PROGRAM PRG_OPT_XPM
VAR
	bInit: BOOL :=TRUE;
	
	fb2AxesXPM: FB_2AxesTrans;
	bExecuteMotionXPM: BOOL :=TRUE;
	bMoveOkXPM: BOOL :=TRUE;
END_VAR

VAR CONSTANT
	rDistance	:REAL	:=	0.4;
END_VAR



IF bINIT THEN
	
	GVL_Main.M12.nBrakeMode := ENUM_StageBrakeMode.NO_BRAKE;
	GVL_Main.M12.bHardwareEnable := TRUE;
	GVL_Main.M12.bPowerSelf := TRUE;
	GVL_Main.M13.nBrakeMode := ENUM_StageBrakeMode.NO_BRAKE;
	GVL_Main.M13.bHardwareEnable := TRUE;
	GVL_Main.M13.bPowerSelf := TRUE;
	
		//
	GVL_Main.M12.nEnableMode := ENUM_StageEnableMode.DURING_MOTION ;
	GVL_Main.M13.nEnableMode := ENUM_StageEnableMode.DURING_MOTION ;

	bINIT := FALSE;
END_IF;

fb2AxesXPM(	i_DevName		:=	'OPT_XPM',
			stFirstAxis		:=	GVL_Main.M12,
			stSecondAxis	:=	GVL_Main.M13,
			bExecuteMotion	:=	bExecuteMotionXPM,
			io_fbFFHWO		:=	GVL_PMPS.io_fbFFHWO,
			fbArbiter		:=	GVL_PMPS.fbArbiter,
			rDistance		:=	rDistance,//0.4, // 0.4m
			bMoveOk			:= bMoveOkXPM
);

END_PROGRAM

(* stored: Version 1.1.0.1, ProductVersion 3.1.4022.18
   POU PRG_OPT_XPM: Id {22739f85-3eea-4d07-957d-370832f3ada0}, SpecialFunc None *)
